// TIA Portal V20 export
TYPE "LConSMC_typeInternalDynamics"
// stored: Access Published
   STRUCT
      acceleration : Real := -1.0;   // Acceleration value : Units are taken from the TO
      deceleration : Real := -1.0;   // Deceleration value: Units are taken from the TO
      jerk : Real := -1.0;   // Jerk value : Units are taken from the TO
      abortAcceleration : Bool := FALSE;   // TRUE: Abort acceleration immediately, FALSE: Reduce current acceleration via Jerk
   END_STRUCT;
END_TYPE
